// TIA Portal V20 export
DATA_BLOCK "Hmi"   // DB4
// stored: MemoryReserve 100
   VAR
      mainHeader : Array[0.."NO_OF_PANELS"] of "LAF_typeHeader";   // Input from the status bar of the HMI
      operationInterlock : "LAF_typeOperationInterlockInterface";
   END_VAR
BEGIN
   mainHeader[0].plcToHmi.modeRequestsButtons.visibility := 16#0;
   mainHeader[0].plcToHmi.specialFunctionButtons.visibility := 16#0071_FFFF;
   mainHeader[0].plcToHmi.specialFunctionButtons.operatorControlAllowed := 16#0;
   mainHeader[0].plcToHmi.specialFunctionButtons.active := 16#0;
END_DATA_BLOCK
